KUKA KRL data list: Test1.dat

&ACCESS RVO1
&COMMENT Modul (src/dat) with INI line and PTP HOME at start and end of Program
DEFDAT Test1 PUBLIC

DECL INT mode = 1
DECL BOOL ready = FALSE

DECL E6POS P_A = {X 3, Y 3, Z 4, A 0, B 0, C 0}
DECL E6POS P_B = {X -2, Y -2, Z -4, A 0, B 0, C 0}
DECL E6POS P_C = {X 1, Y 1, Z 0, A 0, B 0, C 0}
DECL E6POS P_D = {X 3, Y 4, Z 1, A 0, B 0, C 0}

DECL FRAME TOOL_DATA[1]
TOOL_DATA[1] = {X 0, Y 0, Z 200, A 0, B 0, C 0}

;FOLD EXTERNAL DECLARATIONS;%{PE}%MKUKATPBASIS,%CEXT,%VCOMMON,%P
;FOLD BASISTECH EXT;%{PE}%MKUKATPBASIS,%CEXT,%VEXT,%P
EXT  BAS (BAS_COMMAND  :IN,REAL  :IN )
DECL INT SUCCESS
;ENDFOLD (BASISTECH EXT)
;FOLD USER EXT;%{E}%MKUKATPUSER,%CEXT,%VEXT,%P
;Make here your modifications

;ENDFOLD (USER EXT)
;ENDFOLD (EXTERNAL DECLERATIONS)
ENDDAT
